FUNCTION_BLOCK FB_Buffer

VAR
	BlankBuffer : ARRAY[1..GVL.Buffer_Size] OF BOOL; //Empty Buffer (placeholder array used for comparison)
	FullBuffer  : ARRAY[1..GVL.Buffer_Size] OF BOOL; //Full Buffer (placeholder array used for comparison)
	
	IsEmpty 	: BOOL; //TRUE if Buffer EMPTY (all part slots available)
	IsFull  	: BOOL; //TRUE if Buffer FULL (no available part slots)
	
	Init_Conf   : BOOL := TRUE; //Initialize Bit for Buffer Configuration
	
	TargetPosition_Buffer : INT;  // Position in X axis of Buffer 
END_VAR


VAR PERSISTENT
	Buffer_Slots        : ARRAY[1..GVL.Buffer_Size] OF BOOL; (*Buffer Slots state; if ARRAY[Index] = TRUE there is part 
																	               if ARRAY[Index] = FALSE part slot is empty *)
	Parts_Serial_Number : ARRAY[1..GVL.Buffer_Size] OF UDINT; (*Parts Serial Number; each part in Buffer is asociated with respective Serial Number
																					tracked from casssete all way to the carrier *)
END_VAR

IF Init_Conf THEN 
	MEMSET(ADR(FullBuffer),16#1,SIZEOF(FullBuffer)); //FullBuffer has all slots TRUE; to be used to compare with actual Buffer Places
Init_Conf := FALSE;
END_IF

IsEmpty := MEMCMP(ADR(BlankBuffer),ADR(Buffer_Slots),SIZEOF(BlankBuffer)) = 0; //TRUE if Buffer has zero parts (all slots are empty)

IsFull := MEMCMP(ADR(FullBuffer),ADR(Buffer_Slots),SIZEOF(FullBuffer)) = 0;  //TRUE if Buffer is full (has zero available slots)

METHOD M_ClearBuffer : BOOL
VAR_INPUT
END_VAR

VAR 
	 i : INT;
END_VAR
//Clears all Buffer Slots from parts 
FOR i := 1 TO GVL.Buffer_Size DO 
	Buffer_Slots[i] := FALSE;
END_FOR
END_METHOD

METHOD PUBLIC M_Find_First_Empty_Pos : INT

VAR 
	 i : INT;
END_VAR
//If not zero, it outputs first available empty buffer slot
FOR i := 1 TO GVL.Buffer_Size DO
    IF NOT Buffer_Slots[i] THEN
        M_Find_First_Empty_Pos := i;
        RETURN;
    END_IF
END_FOR
M_Find_First_Empty_Pos := 0;
END_METHOD

METHOD PUBLIC M_Find_First_Occupied_Pos : INT

VAR 
	 i : INT;
END_VAR
//If not zero, it outputs first available occupied buffer slot
FOR i := 1 TO GVL.Buffer_Size DO
    IF  Buffer_Slots[i] THEN
        M_Find_First_Occupied_Pos := i;
        RETURN;
    END_IF
END_FOR
M_Find_First_Occupied_Pos := 0;
END_METHOD

METHOD M_MoveToPos : BOOL
VAR_INPUT
END_VAR
// This call sends the desired X Buffer Coordinate for part pick/place for picker_2/picker_1 respectively
END_METHOD

METHOD PUBLIC M_PickPartFromBuffer : BOOL
VAR_INPUT
	Select_Index : INT;
END_VAR
//Picker_2 is picking part from Buffer Slot at position Select_Index
Buffer_Slots[Select_Index] := FALSE;
END_METHOD

METHOD M_PlacePartInBuffer : BOOL
VAR_INPUT
	Select_Index       : UINT;
	Part_Serial_Number : UDINT;
END_VAR
//Picker_1 is placing part in Buffer Slot at position Select_Index
Buffer_Slots[Select_Index] := TRUE;
Parts_Serial_Number[Select_Index] := Part_Serial_Number;
END_METHOD

PROPERTY P_TargetPosition_Buffer : INT
GET
P_TargetPosition_Buffer := TargetPosition_Buffer;
END_GET
SET
TargetPosition_Buffer := P_TargetPosition_Buffer;
END_SET
END_PROPERTY

END_FUNCTION_BLOCK

(* stored: Version 1.1.0.1, ProductVersion 3.1.4024.12
   POU FB_Buffer: Id {b4aa607f-9d94-4d0a-a8e1-b05f46e7ae4a}, SpecialFunc None
   Folder Methods: Id {8d888077-65c4-4b4a-aed3-5283654be573}
   Folder Public: Id {8a8667d8-c502-46ba-9706-bd6556207911}
   Method M_ClearBuffer: Id {b6ac521c-be4d-46de-b385-0b949ba5f652}
   Method M_Find_First_Empty_Pos: Id {715b6a9c-f49c-4f6c-be8c-49094d2f2a8d}
   Method M_Find_First_Occupied_Pos: Id {868e29bc-331d-4a14-8fc5-450054de381a}
   Method M_MoveToPos: Id {087dacf1-2a88-46ec-a7b8-aaa5fdd635cc}
   Method M_PickPartFromBuffer: Id {bfdb16f4-87e3-49fb-9c55-85ec6bdc087a}
   Method M_PlacePartInBuffer: Id {8d6c9ac0-d716-45f6-ab80-315fa0726efc}
   Property P_TargetPosition_Buffer: Id {3afd0690-864f-4124-aa8d-b5d4766c332d}
   Get Get: Id {40849e13-26e8-4b49-ba4e-5a7ab56967e1}
   Set Set: Id {9eef446b-52aa-4d24-8fe0-259a79833bb2} *)
